// TwinCAT 3 PLC project Test2_PLC
// ProgramVersion: 3.1.4023.0
// libraries:
//   Tc2_Standard, * (Beckhoff Automation GmbH)
//   Tc2_System, * (Beckhoff Automation GmbH)
//   Tc3_Module, * (Beckhoff Automation GmbH)
// project tree:
//   GVLs/ GVL.TcGVL
//   / PlcTask.TcTTO
//   POUs/ MAIN.TcPOU
// real-time tasks:
//   TASK PlcTask: cycle T#10ms, priority 20, ADS port 350

CONFIGURATION Test2_PLC
    RESOURCE PLC ON TwinCAT3
        TASK PlcTask(INTERVAL := T#10ms, PRIORITY := 20);
        PROGRAM MAIN WITH PlcTask : MAIN;
    END_RESOURCE
END_CONFIGURATION

// ---- GVLs/GVL.TcGVL
{attribute 'qualified_only'}
VAR_GLOBAL
	nTestValue			: INT;
END_VAR

// ---- POUs/MAIN.TcPOU
PROGRAM MAIN
VAR
	fTestReal		: REAL;
	bTestBool		: BOOL;
	nCycleTime		: UDINT;
	nCycleTime_ms	: INT;
	nTime			: INT;
	nPeriod_ms		: INT;
	nAmplitude		: INT;
	
	fbGetCurTaskIndex	: GETCURTASKINDEX;
END_VAR

fbGetCurTaskIndex();
nCycleTime := _TaskInfo[fbGetCurTaskIndex.index].CycleTime;
nCycleTime_ms := UDINT_TO_INT(nCycleTime/10000);

//Set Sinusoid Amplitude and Period
nAmplitude := 100;
nPeriod_ms := 10000;

//Do 1 sinusoid per second
nTime := (nTime + nCycleTime_ms) MOD nPeriod_ms;

fTestReal := INT_TO_REAL(nAmplitude)*SIN(2*PI*INT_TO_REAL(nTime)/INT_TO_REAL(nPeriod_ms));

GVL.nTestValue := REAL_TO_INT(fTestReal);

END_PROGRAM
